(* IEC 61131-3 sources: FB_Sequence/tests, 8 files *)

(* ---- FB_SEQ_ControlMock.st ---- *)
// OFFLINE TEST DOUBLE ONLY. No I/O, equipment logic or safety function.
// Call before FB_Sequence in the same cyclic task: requests take one scan to echo.
FUNCTION_BLOCK FB_SEQ_ControlMock
VAR_INPUT
    xEnable : BOOL := FALSE;
    stRequest : ST_SEQ_CONTROL_REQUEST;
    stConfig : ST_SEQ_CONFIG;
    xAllowRequests : BOOL := FALSE;
    xAllowExecution : BOOL := FALSE;
    xAllowPublication : BOOL := FALSE;
    xQualified : BOOL := FALSE;
    xStepComplete : BOOL := FALSE;
    xFaulted : BOOL := FALSE;
    xRejectRequest : BOOL := FALSE;
    xFinishActions : BOOL := FALSE;
    udiAuthorityID : UDINT := 0;
END_VAR
VAR_OUTPUT
    stAuthority : ST_SEQ_CONTROL_AUTHORITY;
    stResult : ST_SEQ_CONTROL_RESULT;
    stRuntime : ST_SEQ_CONTROL_RUNTIME;
END_VAR
VAR
    stEmptyAuthority : ST_SEQ_CONTROL_AUTHORITY;
    stEmptyResult : ST_SEQ_CONTROL_RESULT;
    stEmptyRuntime : ST_SEQ_CONTROL_RUNTIME;
    xGrantValid : BOOL;
    xRequestMatches : BOOL;
    xOwnerMatches : BOOL;
    xOwned : BOOL;
    xClosureDone : BOOL;
    udiOwnerSession : UDINT;
    uiOwnerProcess : UINT;
    udiOwnerBatch : UDINT;
    udiToken : UDINT;
END_VAR

// Permission loss, disable and authority epoch changes NEVER release ownership.
// Reinitialize this non-retained test instance to reset the entire mock.
stAuthority := stEmptyAuthority;
stResult := stEmptyResult;
stRuntime := stEmptyRuntime;
xGrantValid := xEnable AND (stConfig.udiSessionID > 0)
    AND (stConfig.uiProcessID > 0) AND (udiAuthorityID > 0);
IF xGrantValid THEN
    stAuthority.xValid := TRUE;
    stAuthority.udiSessionID := stConfig.udiSessionID;
    stAuthority.uiProcessID := stConfig.uiProcessID;
    stAuthority.udiAuthorityID := udiAuthorityID;
    stAuthority.udiAgeMs := 0; // Freshly republished on every invocation.
    stAuthority.xAllowRequests := xAllowRequests;
    stAuthority.xAllowExecution := xAllowExecution;
    stAuthority.xAllowPublication := xAllowPublication;

    stRuntime.xValid := TRUE;
    stRuntime.udiSessionID := stConfig.udiSessionID;
    stRuntime.uiProcessID := stConfig.uiProcessID;
    stRuntime.udiAuthorityID := udiAuthorityID;
    stRuntime.udiAgeMs := 0;
    stRuntime.xReady := NOT xFaulted;
    stRuntime.xFaulted := xFaulted;
    stRuntime.udiBatchID := udiOwnerBatch;
END_IF;

xRequestMatches := xGrantValid AND xAllowRequests AND stRequest.xValid
    AND (stRequest.udiSessionID = stConfig.udiSessionID)
    AND (stRequest.uiProcessID = stConfig.uiProcessID)
    AND (stRequest.udiAuthorityID = udiAuthorityID)
    AND (stRequest.udiBatchID > 0) AND (stRequest.udiIntentID > 0);
xOwnerMatches := (stRequest.udiSessionID = udiOwnerSession)
    AND (stRequest.uiProcessID = uiOwnerProcess)
    AND (stRequest.udiBatchID = udiOwnerBatch);

IF xRequestMatches THEN
    stResult.xValid := TRUE;
    stResult.udiSessionID := stRequest.udiSessionID;
    stResult.uiProcessID := stRequest.uiProcessID;
    stResult.udiAuthorityID := stRequest.udiAuthorityID;
    stResult.udiBatchID := stRequest.udiBatchID;
    stResult.udiIntentID := stRequest.udiIntentID;
    stResult.udiAgeMs := 0;
    stRuntime.udiBatchID := stRequest.udiBatchID;
    stRuntime.udiIntentID := stRequest.udiIntentID;
    // Explicit positive handling below; unsupported requests are rejected.
    IF NOT xRejectRequest THEN
        CASE stRequest.eAction OF
        E_SEQ_ACTION.Acquire:
            IF xAllowExecution AND NOT xFaulted AND ((NOT xOwned) OR xOwnerMatches) THEN
                IF NOT xOwned THEN
                    xOwned := TRUE;
                    udiOwnerSession := stRequest.udiSessionID;
                    uiOwnerProcess := stRequest.uiProcessID;
                    udiOwnerBatch := stRequest.udiBatchID;
                    udiToken := 1;
                    xClosureDone := FALSE;
                END_IF;
                stResult.xAccepted := TRUE;
                stResult.xDone := TRUE;
            END_IF;
        E_SEQ_ACTION.Execute:
            IF xAllowExecution AND NOT xFaulted AND xOwned AND xOwnerMatches
               AND (stRequest.udiResourceToken = udiToken) THEN
                stResult.xAccepted := TRUE;
                stRuntime.xQualified := xQualified;
                stRuntime.xStepComplete := xStepComplete;
                // Acceptance never implies step completion or a lifecycle Done.
                xClosureDone := FALSE;
            END_IF;
        E_SEQ_ACTION.Hold:
            IF xOwned AND xOwnerMatches AND (stRequest.udiResourceToken = udiToken) THEN
                stResult.xAccepted := TRUE;
                stResult.xDone := xFinishActions;
                xClosureDone := FALSE; // A confirmed hold is not batch closure.
            END_IF;
        E_SEQ_ACTION.Complete, E_SEQ_ACTION.Stop, E_SEQ_ACTION.Abort:
            IF (NOT xOwned) OR xOwnerMatches THEN
                // Token zero may occur if an Acquire ACK was lost before abort.
                // Session/process/batch still identify the owned transaction.
                stResult.xAccepted := TRUE;
                stResult.xDone := xFinishActions;
                IF xFinishActions THEN
                    xClosureDone := TRUE;
                    udiOwnerSession := stRequest.udiSessionID;
                    uiOwnerProcess := stRequest.uiProcessID;
                    udiOwnerBatch := stRequest.udiBatchID;
                END_IF;
            END_IF;
        E_SEQ_ACTION.Release:
            IF xOwnerMatches AND xClosureDone THEN
                stResult.xAccepted := TRUE;
                stResult.xDone := TRUE;
                xOwned := FALSE;
                udiToken := 0;
                // Preserve closed identity for idempotent repeated Release.
                stResult.xReleased := TRUE;
            END_IF;
        END_CASE;
    END_IF;
    stResult.xRejected := NOT stResult.xAccepted;
    IF stResult.xRejected THEN stResult.uiReasonID := 1; END_IF;
    stResult.xResourceGranted := xOwned;
    stResult.udiResourceToken := udiToken;
END_IF;

IF xGrantValid THEN
    stRuntime.xResourceGranted := xOwned;
    stRuntime.udiResourceToken := udiToken;
END_IF;
END_FUNCTION_BLOCK

(* ---- PRG_SEQ_AuthorityTests.st ---- *)
// OFFLINE CORRELATION REGRESSION, 8 scans. Expected TRUE,8,0,65535 for
// xDone,uiChecks,uiFailures,uiFirstFailureStep. Requires target IDE execution.
// A Release result from authority 1 cannot combine with runtime from authority 2.
PROGRAM PRG_SEQ_AuthorityTests
VAR
    fbSeq : FB_Sequence;
    fbMock : FB_SEQ_ControlMock;
    stConfig : ST_SEQ_CONFIG;
    stRecipe : ST_SEQ_RECIPE;
    stCommand : ST_SEQ_COMMAND_REQUEST;
    stAuthorityToSeq : ST_SEQ_CONTROL_AUTHORITY;
    stRuntimeToSeq : ST_SEQ_CONTROL_RUNTIME;
    udiAuthorityID : UDINT := 1;
    udiReleaseIntentBefore : UDINT;
    xAllowExecution : BOOL := TRUE;
    xFinishActions : BOOL;
    xPass : BOOL;
    uiStep : UINT;
    uiChecks : UINT;
    uiFailures : UINT;
    uiFirstFailureStep : UINT := UINT#65535;
    xDone : BOOL;
END_VAR

IF xDone THEN RETURN; END_IF;
stCommand.xValid := FALSE;
xFinishActions := FALSE;
CASE uiStep OF
0:
    stConfig.uiProcessID := 1;
    stConfig.udiSessionID := 6001;
    stConfig.udiMaxFeedbackAgeMs := 100;
    stConfig.udiTransitionTimeoutMs := 1000;
    stConfig.udiMaxCycleMs := 100;
    stRecipe.udiRecipeID := 10;
    stRecipe.udiRevision := 1;
    stRecipe.uiStepCount := 1;
    stRecipe.astSteps[1].uiStepID := 100;
    stRecipe.astSteps[1].uiPhaseID := 1;
    stRecipe.astSteps[1].uiProfileID := 1;
    stRecipe.astSteps[1].eKind := E_SEQ_STEP_KIND.WaitComplete;
    stRecipe.astSteps[1].udiTimeoutMs := 5000;
    stCommand.udiSessionID := stConfig.udiSessionID;
    stCommand.uiProcessID := 1;
    stCommand.uiSourceID := 1;
    stCommand.udiRecipeID := 10;
    stCommand.udiRecipeRevision := 1;
    stCommand.udiRequestID := 1;
    stCommand.eCommand := E_SEQ_CMD.LoadRecipe;
    stCommand.xValid := TRUE;
1:
    stCommand.udiBatchID := 1;
    stCommand.udiRequestID := 2;
    stCommand.eCommand := E_SEQ_CMD.Start;
    stCommand.xValid := TRUE;
3:
    xAllowExecution := FALSE;
4:
    xFinishActions := TRUE;
5:
    udiReleaseIntentBefore := fbSeq.stControlRequest.udiIntentID;
6:
    udiAuthorityID := 2;
7:
    stCommand.udiRequestID := 3;
    stCommand.eCommand := E_SEQ_CMD.Reset;
    stCommand.xValid := TRUE;
END_CASE;
fbMock(xEnable := TRUE, stRequest := fbSeq.stControlRequest,
    stConfig := stConfig, xAllowRequests := TRUE,
    xAllowExecution := xAllowExecution, xAllowPublication := TRUE,
    xQualified := FALSE, xStepComplete := FALSE,
    xFaulted := FALSE, xRejectRequest := FALSE,
    xFinishActions := xFinishActions, udiAuthorityID := udiAuthorityID);
stAuthorityToSeq := fbMock.stAuthority;
stRuntimeToSeq := fbMock.stRuntime;
IF uiStep = 5 THEN
    // All scalar freshness/BatchID/IntentID fields match, but generations differ.
    // Keep the valid old-generation Release result intact to reproduce the bug.
    stAuthorityToSeq.udiAuthorityID := 2;
    stRuntimeToSeq.udiAuthorityID := 2;
END_IF;
fbSeq(xEnable := TRUE, stConfig := stConfig, udiDeltaMs := 10,
    stCommand := stCommand, stRecipeCandidate := stRecipe,
    stAuthority := stAuthorityToSeq, stControlResult := fbMock.stResult,
    stControlRuntime := stRuntimeToSeq,
    udiEventAckSessionID := 0, udiEventAckID := 0);
xPass := FALSE;
CASE uiStep OF
0:
    xPass := fbSeq.stRuntime.xRecipeLoaded;
1:
    xPass := fbSeq.stRuntime.eState = E_SEQ_STATE.Starting;
2:
    xPass := fbSeq.stRuntime.eState = E_SEQ_STATE.Running;
3:
    xPass := (fbSeq.stRuntime.eState = E_SEQ_STATE.Faulted)
        AND (fbSeq.stControlRequest.eAction = E_SEQ_ACTION.Abort);
4:
    xPass := (fbSeq.stRuntime.eState = E_SEQ_STATE.Faulted)
        AND (fbSeq.stControlRequest.eAction = E_SEQ_ACTION.Release);
5:
    xPass := fbMock.stResult.xReleased AND (fbMock.stResult.udiAuthorityID = 1)
        AND (fbSeq.stRuntime.eState = E_SEQ_STATE.Faulted)
        AND fbSeq.stControlRequest.xValid
        AND (fbSeq.stControlRequest.eAction = E_SEQ_ACTION.Release)
        AND (fbSeq.stControlRequest.udiAuthorityID = 2)
        AND (fbSeq.stControlRequest.udiIntentID > udiReleaseIntentBefore);
6:
    xPass := fbMock.stResult.xReleased AND (fbMock.stResult.udiAuthorityID = 2)
        AND (fbSeq.stRuntime.eState = E_SEQ_STATE.Faulted)
        AND NOT fbSeq.stControlRequest.xValid;
7:
    xPass := (fbSeq.stRuntime.eState = E_SEQ_STATE.Idle)
        AND (fbSeq.stCommandResult.eResult = E_SEQ_RESULT.Accepted);
END_CASE;
uiChecks := uiChecks + 1;
IF NOT xPass THEN
    uiFailures := uiFailures + 1;
    IF uiFirstFailureStep = UINT#65535 THEN uiFirstFailureStep := uiStep; END_IF;
END_IF;
IF uiStep >= 7 THEN xDone := TRUE;
ELSE uiStep := uiStep + 1; END_IF;
END_PROGRAM

(* ---- PRG_SEQ_Demo.st ---- *)
PROGRAM PRG_SEQ_Demo
VAR
    // Offline-only sandbox. Both mock and Sequence begin disabled.
    xControlMockEnabled : BOOL := FALSE;
    xSequenceEnabled : BOOL := FALSE;
    xAllowRequests : BOOL := FALSE;
    xAllowExecution : BOOL := FALSE;
    xAllowPublication : BOOL := FALSE;
    xQualified : BOOL := FALSE;
    xStepComplete : BOOL := FALSE;
    xFaulted : BOOL := FALSE;
    xRejectRequest : BOOL := FALSE;
    xFinishActions : BOOL := FALSE;
    udiAuthorityID : UDINT := 1;
    stConfig : ST_SEQ_CONFIG := (uiProcessID := 1, udiSessionID := 1,
        udiMaxFeedbackAgeMs := 250, udiTransitionTimeoutMs := 5000, udiMaxCycleMs := 100);
    stCommand : ST_SEQ_COMMAND_REQUEST;
    stRecipe : ST_SEQ_RECIPE;
    udiAckSessionID : UDINT;
    udiAckEventID : UDINT;
    fbControlMock : FB_SEQ_ControlMock;
    fbSequence : FB_Sequence;
    xInitialized : BOOL;
END_VAR

IF NOT xInitialized THEN
    xInitialized := TRUE;
    stRecipe.udiRecipeID := 1;
    stRecipe.udiRevision := 1;
    stRecipe.uiStepCount := 3;
    stRecipe.astSteps[1].uiStepID := 10;
    stRecipe.astSteps[1].uiPhaseID := 10;
    stRecipe.astSteps[1].uiProfileID := 100;
    stRecipe.astSteps[1].eKind := E_SEQ_STEP_KIND.WaitQualified;
    stRecipe.astSteps[1].udiQualifiedMs := 250;
    stRecipe.astSteps[1].udiTimeoutMs := 10000;
    stRecipe.astSteps[2].uiStepID := 20;
    stRecipe.astSteps[2].uiPhaseID := 20;
    stRecipe.astSteps[2].uiProfileID := 200;
    stRecipe.astSteps[2].eKind := E_SEQ_STEP_KIND.WaitComplete;
    stRecipe.astSteps[2].udiTimeoutMs := 10000;
    stRecipe.astSteps[3].uiStepID := 30;
    stRecipe.astSteps[3].uiPhaseID := 30;
    stRecipe.astSteps[3].uiProfileID := 300;
    stRecipe.astSteps[3].eKind := E_SEQ_STEP_KIND.WaitOperator;
    stRecipe.astSteps[3].udiTimeoutMs := 10000;
END_IF;

// One task, one call per scan, previous request consumed by mock on next scan.
fbControlMock(xEnable := xControlMockEnabled, stRequest := fbSequence.stControlRequest,
    stConfig := stConfig, xAllowRequests := xAllowRequests, xAllowExecution := xAllowExecution,
    xAllowPublication := xAllowPublication, xQualified := xQualified,
    xStepComplete := xStepComplete, xFaulted := xFaulted, xRejectRequest := xRejectRequest,
    xFinishActions := xFinishActions, udiAuthorityID := udiAuthorityID);
fbSequence(xEnable := xSequenceEnabled, stConfig := stConfig, udiDeltaMs := 20,
    stCommand := stCommand, stRecipeCandidate := stRecipe,
    stAuthority := fbControlMock.stAuthority, stControlResult := fbControlMock.stResult,
    stControlRuntime := fbControlMock.stRuntime,
    udiEventAckSessionID := udiAckSessionID, udiEventAckID := udiAckEventID);
// 20 ms here is synthetic simulation time, not a claim of measured target timing.
END_PROGRAM

(* ---- PRG_SEQ_IntegrationTests.st ---- *)
// OFFLINE MULTISCAN TEST POU: import with production types/FBs and ControlMock.
// Assign ONLY to a simulator/test task with no physical I/O. Every call is 10 ms
// of simulated time. Fresh non-retained instances run 28 checks in 28 calls.
// Inspect xDone, uiChecks, uiFailures, uiFirstFailureStep. Expected: TRUE,28,0,65535.
// Reinitialize the application to rerun; changing uiStep alone is insufficient.
// These are executable IDE test scenarios; their presence is not a test-run claim.
PROGRAM PRG_SEQ_IntegrationTests
VAR
    fbSeq : FB_Sequence;
    fbMock : FB_SEQ_ControlMock;
    stConfig : ST_SEQ_CONFIG;
    stRecipe : ST_SEQ_RECIPE;
    stCommand : ST_SEQ_COMMAND_REQUEST;
    stResultToSeq : ST_SEQ_CONTROL_RESULT;
    stRuntimeToSeq : ST_SEQ_CONTROL_RUNTIME;
    xMockEnable : BOOL;
    xAllowRequests : BOOL;
    xAllowExecution : BOOL;
    xAllowPublication : BOOL;
    xQualified : BOOL;
    xStepComplete : BOOL;
    xFinishActions : BOOL;
    udiAuthorityID : UDINT;
    xCorruptResultID : BOOL;
    xCorruptRuntimeID : BOOL;
    xPass : BOOL;
    uiStep : UINT;
    uiChecks : UINT;
    uiFailures : UINT;
    uiFirstFailureStep : UINT := UINT#65535;
    xDone : BOOL;
END_VAR

IF xDone THEN RETURN; END_IF;

// Default stimuli are inert; permission changes remain in effect across scans.
stCommand.xValid := FALSE;
xQualified := FALSE;
xStepComplete := FALSE;
xFinishActions := FALSE;
xCorruptResultID := FALSE;
xCorruptRuntimeID := FALSE;

CASE uiStep OF
0: // Neither mock enable nor a Control grant exists.
    stConfig.uiProcessID := 1;
    stConfig.udiSessionID := 1001;
    stConfig.udiMaxFeedbackAgeMs := 100;
    stConfig.udiTransitionTimeoutMs := 1000;
    stConfig.udiMaxCycleMs := 100;
    stRecipe.udiRecipeID := 10;
    stRecipe.udiRevision := 1;
    stRecipe.uiStepCount := 1;
    stRecipe.astSteps[1].uiStepID := 100;
    stRecipe.astSteps[1].uiPhaseID := 1;
    stRecipe.astSteps[1].uiProfileID := 1;
    stRecipe.astSteps[1].eKind := E_SEQ_STEP_KIND.WaitQualified;
    stRecipe.astSteps[1].udiQualifiedMs := 30;
    stRecipe.astSteps[1].udiTimeoutMs := 2000;
    stCommand.udiSessionID := stConfig.udiSessionID;
    stCommand.uiProcessID := stConfig.uiProcessID;
    stCommand.uiSourceID := 1;
    stCommand.udiRecipeID := stRecipe.udiRecipeID;
    stCommand.udiRecipeRevision := stRecipe.udiRevision;
    stCommand.udiRequestID := 1;
    stCommand.eCommand := E_SEQ_CMD.LoadRecipe;
    stCommand.xValid := TRUE;
1: // Permission bits alone cannot manufacture a nonzero Control authority.
    xMockEnable := TRUE;
    xAllowRequests := TRUE;
    xAllowExecution := TRUE;
    xAllowPublication := TRUE;
2: // A new request ID is required after the denied request.
    udiAuthorityID := 1;
    stCommand.udiRequestID := 2;
    stCommand.eCommand := E_SEQ_CMD.LoadRecipe;
    stCommand.xValid := TRUE;
3:
    stCommand.udiRequestID := 3;
    stCommand.eCommand := E_SEQ_CMD.Start;
    stCommand.udiBatchID := 1;
    stCommand.xValid := TRUE;
4: // Acquire has completed in Control, but an unrelated ACK cannot advance.
    xCorruptResultID := TRUE;
5: // The original matching Acquire result is now admitted.
    ;
6: // A matching accepted result plus unrelated runtime is still insufficient.
    xQualified := TRUE;
    xStepComplete := TRUE;
    xCorruptRuntimeID := TRUE;
7: // First qualified observation establishes the interval boundary.
    xQualified := TRUE;
8: // An unqualified interval must not accrue qualified time.
    xQualified := FALSE;
9, 10, 11, 12:
    xQualified := TRUE;
13: // Control accepted Complete, but has not finished the physical closure.
    ;
14:
    xFinishActions := TRUE;
15: // Release is a separate transaction after closure Done.
    ;
16:
    stCommand.udiRequestID := 4;
    stCommand.eCommand := E_SEQ_CMD.Reset;
    stCommand.xValid := TRUE;
17:
    stCommand.udiRequestID := 5;
    stCommand.eCommand := E_SEQ_CMD.Start;
    stCommand.udiBatchID := 2;
    stCommand.xValid := TRUE;
18:
    ;
19: // Revoke requests and execution during the second batch.
    xAllowRequests := FALSE;
    xAllowExecution := FALSE;
20: // Restoring both permissions cannot resume the faulted batch.
    xAllowRequests := TRUE;
    xAllowExecution := TRUE;
21: // Publication permission controls every public Service envelope.
    xAllowPublication := FALSE;
22: // Requests remain permitted for closure while execution is denied.
    xAllowPublication := TRUE;
    xAllowExecution := FALSE;
23: // New Control epoch must not silently erase existing ownership.
    udiAuthorityID := 2;
24:
    xFinishActions := TRUE;
25:
    ;
26: // Reset requires the confirmed Abort then Release, not just a new grant.
    stCommand.udiRequestID := 6;
    stCommand.eCommand := E_SEQ_CMD.Reset;
    stCommand.xValid := TRUE;
27: // Request permission does not imply permission to start execution.
    stCommand.udiRequestID := 7;
    stCommand.eCommand := E_SEQ_CMD.Start;
    stCommand.udiBatchID := 3;
    stCommand.xValid := TRUE;
END_CASE;

// One scan of request/feedback latency, with fresh snapshots on every mock call.
fbMock(xEnable := xMockEnable, stRequest := fbSeq.stControlRequest,
    stConfig := stConfig, xAllowRequests := xAllowRequests,
    xAllowExecution := xAllowExecution, xAllowPublication := xAllowPublication,
    xQualified := xQualified, xStepComplete := xStepComplete,
    xFaulted := FALSE, xRejectRequest := FALSE,
    xFinishActions := xFinishActions, udiAuthorityID := udiAuthorityID);
stResultToSeq := fbMock.stResult;
stRuntimeToSeq := fbMock.stRuntime;
IF xCorruptResultID THEN
    stResultToSeq.udiIntentID := stResultToSeq.udiIntentID + 100;
END_IF;
IF xCorruptRuntimeID THEN
    stRuntimeToSeq.udiIntentID := stRuntimeToSeq.udiIntentID + 100;
END_IF;
fbSeq(xEnable := TRUE, stConfig := stConfig, udiDeltaMs := 10,
    stCommand := stCommand, stRecipeCandidate := stRecipe,
    stAuthority := fbMock.stAuthority, stControlResult := stResultToSeq,
    stControlRuntime := stRuntimeToSeq,
    udiEventAckSessionID := 0, udiEventAckID := 0);

xPass := FALSE;
CASE uiStep OF
0, 1:
    xPass := NOT fbSeq.stControlRequest.xValid
        AND NOT fbSeq.stRuntime.xDataValid AND NOT fbSeq.stCommandResult.xValid
        AND NOT fbSeq.xEventAvailable AND (fbSeq.uiEventCount = 0)
        AND (fbSeq.stRuntime.udiSessionID = 0) AND (fbSeq.stEvent.udiEventID = 0);
2:
    xPass := fbSeq.stRuntime.xDataValid AND fbSeq.stRuntime.xRecipeLoaded
        AND (fbSeq.stRuntime.eState = E_SEQ_STATE.Idle)
        AND (fbSeq.stCommandResult.eResult = E_SEQ_RESULT.Accepted)
        AND (fbSeq.stCommandResult.udiRequestID = 2);
3:
    xPass := (fbSeq.stRuntime.eState = E_SEQ_STATE.Starting)
        AND (fbSeq.stControlRequest.eAction = E_SEQ_ACTION.Acquire)
        AND fbSeq.stControlRequest.xValid;
4:
    xPass := fbMock.stResult.xDone AND fbMock.stRuntime.xResourceGranted
        AND (fbSeq.stRuntime.eState = E_SEQ_STATE.Starting)
        AND (fbSeq.stRuntime.udiResourceToken = 0)
        AND (fbSeq.stControlRequest.eAction = E_SEQ_ACTION.Acquire);
5:
    xPass := (fbSeq.stRuntime.eState = E_SEQ_STATE.Running)
        AND (fbSeq.stControlRequest.eAction = E_SEQ_ACTION.Execute)
        AND (fbSeq.stRuntime.udiResourceToken = 1);
6:
    xPass := fbMock.stResult.xAccepted AND NOT fbMock.stResult.xDone
        AND (fbSeq.stRuntime.eState = E_SEQ_STATE.Running)
        AND (fbSeq.stRuntime.udiQualifiedElapsedMs = 0);
7, 8, 9:
    xPass := (fbSeq.stRuntime.eState = E_SEQ_STATE.Running)
        AND (fbSeq.stRuntime.udiQualifiedElapsedMs = 0);
10:
    xPass := (fbSeq.stRuntime.eState = E_SEQ_STATE.Running)
        AND (fbSeq.stRuntime.udiQualifiedElapsedMs = 10);
11:
    xPass := (fbSeq.stRuntime.eState = E_SEQ_STATE.Running)
        AND (fbSeq.stRuntime.udiQualifiedElapsedMs = 20);
12:
    xPass := (fbSeq.stRuntime.eState = E_SEQ_STATE.Completing)
        AND (fbSeq.stControlRequest.eAction = E_SEQ_ACTION.Complete)
        AND (fbSeq.stRuntime.udiQualifiedElapsedMs = 30)
        AND fbMock.stRuntime.xResourceGranted;
13:
    xPass := fbMock.stResult.xAccepted AND NOT fbMock.stResult.xDone
        AND (fbSeq.stRuntime.eState = E_SEQ_STATE.Completing)
        AND (fbSeq.stControlRequest.eAction = E_SEQ_ACTION.Complete)
        AND fbMock.stRuntime.xResourceGranted;
14:
    xPass := fbMock.stResult.xDone
        AND (fbSeq.stRuntime.eState = E_SEQ_STATE.Completing)
        AND (fbSeq.stControlRequest.eAction = E_SEQ_ACTION.Release)
        AND fbMock.stRuntime.xResourceGranted;
15:
    xPass := fbMock.stResult.xReleased AND NOT fbMock.stRuntime.xResourceGranted
        AND (fbSeq.stRuntime.eState = E_SEQ_STATE.Complete)
        AND (fbSeq.stRuntime.udiResourceToken = 0)
        AND NOT fbSeq.stControlRequest.xValid;
16:
    xPass := (fbSeq.stRuntime.eState = E_SEQ_STATE.Idle)
        AND (fbSeq.stRuntime.udiBatchID = 0)
        AND (fbSeq.stCommandResult.eResult = E_SEQ_RESULT.Accepted);
17:
    xPass := (fbSeq.stRuntime.eState = E_SEQ_STATE.Starting)
        AND (fbSeq.stRuntime.udiBatchID = 2)
        AND (fbSeq.stControlRequest.eAction = E_SEQ_ACTION.Acquire);
18:
    xPass := (fbSeq.stRuntime.eState = E_SEQ_STATE.Running)
        AND (fbSeq.stControlRequest.eAction = E_SEQ_ACTION.Execute)
        AND fbMock.stRuntime.xResourceGranted;
19:
    xPass := (fbSeq.stRuntime.eState = E_SEQ_STATE.Faulted)
        AND (fbSeq.stRuntime.eReason = E_SEQ_REASON.AuthorityDenied)
        AND NOT fbSeq.stControlRequest.xValid AND NOT fbMock.stResult.xValid
        AND fbMock.stRuntime.xResourceGranted;
20:
    xPass := (fbSeq.stRuntime.eState = E_SEQ_STATE.Faulted)
        AND fbSeq.stControlRequest.xValid
        AND (fbSeq.stControlRequest.eAction = E_SEQ_ACTION.Abort)
        AND fbMock.stRuntime.xResourceGranted;
21:
    xPass := NOT fbSeq.stRuntime.xDataValid AND NOT fbSeq.stCommandResult.xValid
        AND (fbSeq.stRuntime.udiSessionID = 0) AND (fbSeq.stRuntime.udiBatchID = 0)
        AND (fbSeq.stCommandResult.udiRequestID = 0)
        AND NOT fbSeq.xEventAvailable AND (fbSeq.stEvent.udiEventID = 0)
        AND (fbSeq.uiEventCount = 0) AND (fbSeq.udiEventsDropped = 0)
        AND (fbSeq.stControlRequest.eAction = E_SEQ_ACTION.Abort)
        AND fbMock.stRuntime.xResourceGranted;
22:
    xPass := (fbSeq.stRuntime.eState = E_SEQ_STATE.Faulted)
        AND (fbSeq.stControlRequest.eAction = E_SEQ_ACTION.Abort)
        AND fbSeq.xEventAvailable AND fbMock.stRuntime.xResourceGranted;
23:
    xPass := (fbSeq.stRuntime.eState = E_SEQ_STATE.Faulted)
        AND (fbSeq.stControlRequest.eAction = E_SEQ_ACTION.Abort)
        AND (fbSeq.stControlRequest.udiAuthorityID = 2)
        AND NOT fbMock.stResult.xValid AND fbMock.stRuntime.xResourceGranted;
24:
    xPass := (fbSeq.stRuntime.eState = E_SEQ_STATE.Faulted)
        AND fbMock.stResult.xDone AND (fbSeq.stControlRequest.eAction = E_SEQ_ACTION.Release)
        AND fbMock.stRuntime.xResourceGranted;
25:
    xPass := (fbSeq.stRuntime.eState = E_SEQ_STATE.Faulted)
        AND fbMock.stResult.xReleased AND NOT fbMock.stRuntime.xResourceGranted
        AND NOT fbSeq.stControlRequest.xValid AND (fbSeq.stRuntime.udiResourceToken = 0);
26:
    xPass := (fbSeq.stRuntime.eState = E_SEQ_STATE.Idle)
        AND (fbSeq.stCommandResult.eResult = E_SEQ_RESULT.Accepted)
        AND NOT fbMock.stRuntime.xResourceGranted;
27:
    xPass := (fbSeq.stRuntime.eState = E_SEQ_STATE.Idle)
        AND (fbSeq.stCommandResult.eResult = E_SEQ_RESULT.Rejected)
        AND (fbSeq.stCommandResult.eReason = E_SEQ_REASON.AuthorityDenied)
        AND NOT fbSeq.stControlRequest.xValid;
END_CASE;

uiChecks := uiChecks + 1;
IF NOT xPass THEN
    IF uiFailures = 0 THEN uiFirstFailureStep := uiStep; END_IF;
    uiFailures := uiFailures + 1;
END_IF;
IF uiStep = 27 THEN xDone := TRUE;
ELSE uiStep := uiStep + 1; END_IF;
END_PROGRAM

(* ---- PRG_SEQ_LifecycleTests.st ---- *)
// OFFLINE MULTISCAN TEST ONLY: no physical I/O or task scheduling assumptions.
// Run a fresh, non-retained instance for 56 simulated scans of 10 ms each.
// Expected: xDone=TRUE, uiChecks=56, uiFailures=0, uiFirstFailureStep=65535.
// Exercises actual FB_Sequence code when run in the target IDE; NOT run here.
PROGRAM PRG_SEQ_LifecycleTests
VAR
    fbSeq : FB_Sequence;
    fbMock : FB_SEQ_ControlMock;
    stConfig : ST_SEQ_CONFIG;
    stRecipe : ST_SEQ_RECIPE;
    stCommand : ST_SEQ_COMMAND_REQUEST;
    stRuntimeToSeq : ST_SEQ_CONTROL_RUNTIME;
    xQualified : BOOL;
    xFinishActions : BOOL;
    xInjectHoldQualified : BOOL;
    xInjectNotReady : BOOL;
    xPass : BOOL;
    xSawResetBatch : BOOL;
    udiRequestID : UDINT;
    udiAck : UDINT;
    udiPrompt : UDINT;
    uiStep : UINT;
    uiChecks : UINT;
    uiFailures : UINT;
    uiFirstFailureStep : UINT := UINT#65535;
    xDone : BOOL;
END_VAR

IF xDone THEN RETURN; END_IF;
stCommand.xValid := FALSE;
xQualified := TRUE;
xFinishActions := FALSE;
xInjectHoldQualified := FALSE;
xInjectNotReady := FALSE;

CASE uiStep OF
0:
    stConfig.uiProcessID := 1;
    stConfig.udiSessionID := 5001;
    stConfig.udiMaxFeedbackAgeMs := 100;
    stConfig.udiTransitionTimeoutMs := 30;
    stConfig.udiMaxCycleMs := 100;
    stRecipe.udiRecipeID := 10;
    stRecipe.udiRevision := 1;
    stRecipe.uiStepCount := 1;
    stRecipe.astSteps[1].uiStepID := 100;
    stRecipe.astSteps[1].uiPhaseID := 1;
    stRecipe.astSteps[1].uiProfileID := 1;
    stRecipe.astSteps[1].eKind := E_SEQ_STEP_KIND.WaitQualified;
    stRecipe.astSteps[1].udiQualifiedMs := 100;
    stRecipe.astSteps[1].udiTimeoutMs := 5000;
    stCommand.udiSessionID := stConfig.udiSessionID;
    stCommand.uiProcessID := stConfig.uiProcessID;
    stCommand.uiSourceID := 1;
    stCommand.udiRecipeID := 10;
    stCommand.udiRecipeRevision := 1;
    stCommand.eCommand := E_SEQ_CMD.LoadRecipe;
    stCommand.xValid := TRUE;
1:
    stCommand.udiBatchID := 1;
    stCommand.eCommand := E_SEQ_CMD.Start;
    stCommand.xValid := TRUE;
5:
    stCommand.eCommand := E_SEQ_CMD.Hold;
    stCommand.xValid := TRUE;
6:
    xFinishActions := TRUE;
7:
    xInjectHoldQualified := TRUE;
8: // Old Hold feedback must not qualify the first interval after Resume.
    xInjectHoldQualified := TRUE;
    stCommand.eCommand := E_SEQ_CMD.Resume;
    stCommand.xValid := TRUE;
9: // Changing the candidate cannot mutate the already applied recipe snapshot.
    stRecipe.udiRevision := 99;
    stRecipe.astSteps[1].udiQualifiedMs := 1;
11:
    stCommand.eCommand := E_SEQ_CMD.Stop;
    stCommand.xValid := TRUE;
13:
    xFinishActions := TRUE;
15:
    stCommand.eCommand := E_SEQ_CMD.Reset;
    stCommand.xValid := TRUE;
16:
    stRecipe.udiRevision := 2;
    stRecipe.astSteps[1].eKind := E_SEQ_STEP_KIND.WaitOperator;
    stRecipe.astSteps[1].udiQualifiedMs := 0;
    stCommand.udiRecipeRevision := 2;
    stCommand.eCommand := E_SEQ_CMD.LoadRecipe;
    stCommand.xValid := TRUE;
17:
    stCommand.udiBatchID := 2;
    stCommand.eCommand := E_SEQ_CMD.Start;
    stCommand.xValid := TRUE;
19: // Matching/qualified feedback that is not Ready must reject confirmation.
    udiPrompt := fbSeq.stRuntime.udiPromptID;
    stCommand.uiStepID := 100;
    stCommand.udiPromptID := udiPrompt;
    stCommand.eCommand := E_SEQ_CMD.ConfirmStep;
    stCommand.xValid := TRUE;
    xInjectNotReady := TRUE;
20:
    stCommand.udiPromptID := udiPrompt + 1;
    stCommand.eCommand := E_SEQ_CMD.ConfirmStep;
    stCommand.xValid := TRUE;
26: // Running now exceeds the transition limit; new Completing starts at zero.
    stCommand.udiPromptID := udiPrompt;
    stCommand.eCommand := E_SEQ_CMD.ConfirmStep;
    stCommand.xValid := TRUE;
27:
    xFinishActions := TRUE;
29:
    stCommand.eCommand := E_SEQ_CMD.Reset;
    stCommand.xValid := TRUE;
30:
    stCommand.udiBatchID := 3;
    stCommand.eCommand := E_SEQ_CMD.Start;
    stCommand.xValid := TRUE;
32:
    stCommand.eCommand := E_SEQ_CMD.Abort;
    stCommand.xValid := TRUE;
33:
    xFinishActions := TRUE;
35:
    stCommand.eCommand := E_SEQ_CMD.Reset;
    stCommand.xValid := TRUE;
36:
    stCommand.udiBatchID := 4;
    stCommand.eCommand := E_SEQ_CMD.Start;
    stCommand.xValid := TRUE;
38:
    stCommand.eCommand := E_SEQ_CMD.Hold;
    stCommand.xValid := TRUE;
42:
    xFinishActions := TRUE;
44:
    stCommand.eCommand := E_SEQ_CMD.Reset;
    stCommand.xValid := TRUE;
END_CASE;
IF stCommand.xValid THEN
    udiRequestID := udiRequestID + 1;
    stCommand.udiRequestID := udiRequestID;
END_IF;

// Acknowledge ONLY an event actually observed in the previous published scan.
udiAck := 0;
IF fbSeq.xEventAvailable THEN
    udiAck := fbSeq.stEvent.udiEventID;
    IF (fbSeq.stEvent.eKind = E_SEQ_EVENT_KIND.CommandResult)
       AND (fbSeq.stEvent.eCommand = E_SEQ_CMD.Reset)
       AND (fbSeq.stEvent.udiBatchID = 1)
       AND (fbSeq.stEvent.eCommandResult = E_SEQ_RESULT.Accepted) THEN
        xSawResetBatch := TRUE;
    END_IF;
END_IF;
fbMock(xEnable := TRUE, stRequest := fbSeq.stControlRequest,
    stConfig := stConfig, xAllowRequests := TRUE,
    xAllowExecution := TRUE, xAllowPublication := TRUE,
    xQualified := xQualified, xStepComplete := FALSE,
    xFaulted := FALSE, xRejectRequest := FALSE,
    xFinishActions := xFinishActions, udiAuthorityID := 1);
stRuntimeToSeq := fbMock.stRuntime;
IF xInjectHoldQualified THEN stRuntimeToSeq.xQualified := TRUE; END_IF;
IF xInjectNotReady THEN stRuntimeToSeq.xReady := FALSE; END_IF;
fbSeq(xEnable := TRUE, stConfig := stConfig, udiDeltaMs := 10,
    stCommand := stCommand, stRecipeCandidate := stRecipe,
    stAuthority := fbMock.stAuthority, stControlResult := fbMock.stResult,
    stControlRuntime := stRuntimeToSeq,
    udiEventAckSessionID := stConfig.udiSessionID, udiEventAckID := udiAck);

xPass := FALSE;
CASE uiStep OF
0:
    xPass := fbSeq.stRuntime.xRecipeLoaded
        AND (fbSeq.stCommandResult.eResult = E_SEQ_RESULT.Accepted);
1, 17, 30, 36:
    xPass := (fbSeq.stRuntime.eState = E_SEQ_STATE.Starting)
        AND (fbSeq.stControlRequest.eAction = E_SEQ_ACTION.Acquire);
2, 3:
    xPass := (fbSeq.stRuntime.eState = E_SEQ_STATE.Running)
        AND (fbSeq.stRuntime.udiQualifiedElapsedMs = 0);
4:
    xPass := (fbSeq.stRuntime.eState = E_SEQ_STATE.Running)
        AND (fbSeq.stRuntime.udiQualifiedElapsedMs = 10);
5:
    xPass := (fbSeq.stRuntime.eState = E_SEQ_STATE.Holding)
        AND (fbSeq.stRuntime.udiQualifiedElapsedMs = 10);
6, 7:
    xPass := (fbSeq.stRuntime.eState = E_SEQ_STATE.Held)
        AND (fbSeq.stRuntime.udiQualifiedElapsedMs = 10);
8, 9:
    xPass := (fbSeq.stRuntime.eState = E_SEQ_STATE.Running)
        AND (fbSeq.stRuntime.udiQualifiedElapsedMs = 10)
        AND (fbSeq.stRuntime.udiRecipeRevision = 1);
10:
    xPass := (fbSeq.stRuntime.eState = E_SEQ_STATE.Running)
        AND (fbSeq.stRuntime.udiQualifiedElapsedMs = 20);
11, 12:
    xPass := (fbSeq.stRuntime.eState = E_SEQ_STATE.Stopping)
        AND (fbSeq.stControlRequest.eAction = E_SEQ_ACTION.Stop);
13:
    xPass := (fbSeq.stRuntime.eState = E_SEQ_STATE.Stopping)
        AND (fbSeq.stControlRequest.eAction = E_SEQ_ACTION.Release);
14:
    xPass := (fbSeq.stRuntime.eState = E_SEQ_STATE.Stopped)
        AND NOT fbSeq.stControlRequest.xValid;
15, 29, 35, 44:
    xPass := (fbSeq.stRuntime.eState = E_SEQ_STATE.Idle)
        AND (fbSeq.stRuntime.udiBatchID = 0)
        AND (fbSeq.stCommandResult.eResult = E_SEQ_RESULT.Accepted);
16:
    xPass := fbSeq.stRuntime.xRecipeLoaded AND (fbSeq.stRuntime.udiRecipeRevision = 2);
18, 21, 22, 23, 24, 25, 31, 37:
    xPass := (fbSeq.stRuntime.eState = E_SEQ_STATE.Running)
        AND fbSeq.stRuntime.xWaitingOperator AND (fbSeq.stRuntime.udiPromptID > 0);
19, 20:
    xPass := (fbSeq.stRuntime.eState = E_SEQ_STATE.Running)
        AND (fbSeq.stCommandResult.eResult = E_SEQ_RESULT.Rejected)
        AND (fbSeq.stCommandResult.eReason = E_SEQ_REASON.InvalidConfirm);
26:
    xPass := (fbSeq.stRuntime.eState = E_SEQ_STATE.Completing)
        AND (fbSeq.stControlRequest.eAction = E_SEQ_ACTION.Complete)
        AND (fbSeq.stRuntime.udiStateElapsedMs = 0)
        AND (fbSeq.stRuntime.eReason = E_SEQ_REASON.None);
27:
    xPass := (fbSeq.stRuntime.eState = E_SEQ_STATE.Completing)
        AND (fbSeq.stControlRequest.eAction = E_SEQ_ACTION.Release);
28:
    xPass := (fbSeq.stRuntime.eState = E_SEQ_STATE.Complete)
        AND NOT fbSeq.stControlRequest.xValid;
32:
    xPass := (fbSeq.stRuntime.eState = E_SEQ_STATE.Aborting)
        AND (fbSeq.stControlRequest.eAction = E_SEQ_ACTION.Abort);
33:
    xPass := (fbSeq.stRuntime.eState = E_SEQ_STATE.Aborting)
        AND (fbSeq.stControlRequest.eAction = E_SEQ_ACTION.Release);
34:
    xPass := (fbSeq.stRuntime.eState = E_SEQ_STATE.Aborted)
        AND NOT fbSeq.stControlRequest.xValid;
38, 39, 40:
    xPass := (fbSeq.stRuntime.eState = E_SEQ_STATE.Holding)
        AND (fbSeq.stControlRequest.eAction = E_SEQ_ACTION.Hold);
41:
    xPass := (fbSeq.stRuntime.eState = E_SEQ_STATE.Faulted)
        AND (fbSeq.stRuntime.eReason = E_SEQ_REASON.TransitionTimeout)
        AND (fbSeq.stControlRequest.eAction = E_SEQ_ACTION.Abort);
42:
    xPass := (fbSeq.stRuntime.eState = E_SEQ_STATE.Faulted)
        AND (fbSeq.stControlRequest.eAction = E_SEQ_ACTION.Release);
43:
    xPass := (fbSeq.stRuntime.eState = E_SEQ_STATE.Faulted)
        AND NOT fbSeq.stControlRequest.xValid
        AND NOT fbMock.stRuntime.xResourceGranted;
ELSE
    xPass := (fbSeq.stRuntime.eState = E_SEQ_STATE.Idle)
        AND (fbSeq.udiEventsDropped = 0);
END_CASE;
IF uiStep = 55 THEN
    xPass := xPass AND xSawResetBatch AND NOT fbSeq.xEventAvailable;
END_IF;
uiChecks := uiChecks + 1;
IF NOT xPass THEN
    uiFailures := uiFailures + 1;
    IF uiFirstFailureStep = UINT#65535 THEN uiFirstFailureStep := uiStep; END_IF;
END_IF;
IF uiStep >= 55 THEN xDone := TRUE;
ELSE uiStep := uiStep + 1; END_IF;
END_PROGRAM

(* ---- PRG_SEQ_SupportTests.st ---- *)
// Simulator-only self-checking POU; no GVLs, physical I/O, network, or tasks.
// Import DUTs, F_SEQ_AddMs, FB_SEQ_* and this PROGRAM into Machine Expert.
// Attach ONLY this POU to a simulator task; observe xDone, uiChecks, uiFailures.
// Expected result: xDone = TRUE, uiChecks = 40, uiFailures = 0.
// Reset/reinitialize the application to rerun: stateful instances are intentional.
// Deliberate sequential FB calls model scan boundaries with explicit deltas.
// These are authored executable simulator tests; not proof of a native compile.
PROGRAM PRG_SEQ_SupportTests
VAR
    xDone : BOOL;
    uiChecks : UINT;
    uiFailures : UINT;
    fbTimer : FB_SEQ_QualifiedTimer;
    fbRecipe : FB_SEQ_RecipeValidator;
    fbQueue : FB_SEQ_EventQueue;
    fbGate : FB_SEQ_CommandGate;
    stRecipe : ST_SEQ_RECIPE;
    stEvent : ST_SEQ_EVENT;
    stCommand : ST_SEQ_COMMAND_REQUEST;
    uiIndex : UINT;
    udiExpectedID : UDINT;
    xDrainCorrect : BOOL;
END_VAR

IF xDone THEN RETURN; END_IF;

// 01 - Overflow-safe addition, including boundary equality.
uiChecks := uiChecks + 1;
IF F_SEQ_AddMs(UDINT#4294967294, UDINT#1) <> UDINT#4294967295 THEN
    uiFailures := uiFailures + 1;
END_IF;
uiChecks := uiChecks + 1;
IF F_SEQ_AddMs(UDINT#4294967294, UDINT#2) <> UDINT#4294967295 THEN
    uiFailures := uiFailures + 1;
END_IF;
uiChecks := uiChecks + 1;
IF F_SEQ_AddMs(UDINT#4294967295, UDINT#4294967295) <> UDINT#4294967295 THEN
    uiFailures := uiFailures + 1;
END_IF;

// 02 - Qualified timer: reset dominates an enabled/qualified call.
fbTimer(xReset := TRUE, xEnable := TRUE, xQualified := TRUE,
    udiDeltaMs := 100, udiTargetMs := 100);
uiChecks := uiChecks + 1;
IF (fbTimer.udiElapsedMs <> 0) OR fbTimer.xDone THEN
    uiFailures := uiFailures + 1;
END_IF;
fbTimer(xReset := FALSE, xEnable := TRUE, xQualified := TRUE,
    udiDeltaMs := 40, udiTargetMs := 100);
uiChecks := uiChecks + 1;
IF (fbTimer.udiElapsedMs <> 40) OR fbTimer.xDone THEN
    uiFailures := uiFailures + 1;
END_IF;
fbTimer(xReset := FALSE, xEnable := FALSE, xQualified := TRUE,
    udiDeltaMs := 80, udiTargetMs := 100);
uiChecks := uiChecks + 1;
IF (fbTimer.udiElapsedMs <> 40) OR fbTimer.xDone THEN
    uiFailures := uiFailures + 1;
END_IF;
fbTimer(xReset := FALSE, xEnable := TRUE, xQualified := FALSE,
    udiDeltaMs := 80, udiTargetMs := 100);
uiChecks := uiChecks + 1;
IF (fbTimer.udiElapsedMs <> 40) OR fbTimer.xDone THEN
    uiFailures := uiFailures + 1;
END_IF;
fbTimer(xReset := FALSE, xEnable := TRUE, xQualified := TRUE,
    udiDeltaMs := UDINT#4294967295, udiTargetMs := 100);
uiChecks := uiChecks + 1;
IF (fbTimer.udiElapsedMs <> 100) OR NOT fbTimer.xDone THEN
    uiFailures := uiFailures + 1;
END_IF;
fbTimer(xReset := FALSE, xEnable := FALSE, xQualified := FALSE,
    udiDeltaMs := 100, udiTargetMs := 100);
uiChecks := uiChecks + 1;
IF (fbTimer.udiElapsedMs <> 100) OR NOT fbTimer.xDone THEN
    uiFailures := uiFailures + 1;
END_IF;
fbTimer(xReset := TRUE, xEnable := TRUE, xQualified := TRUE,
    udiDeltaMs := 100, udiTargetMs := 100);
uiChecks := uiChecks + 1;
IF (fbTimer.udiElapsedMs <> 0) OR fbTimer.xDone THEN
    uiFailures := uiFailures + 1;
END_IF;
fbTimer(xReset := FALSE, xEnable := TRUE, xQualified := TRUE,
    udiDeltaMs := 100, udiTargetMs := 0);
uiChecks := uiChecks + 1;
IF (fbTimer.udiElapsedMs <> 0) OR fbTimer.xDone THEN
    uiFailures := uiFailures + 1;
END_IF;

// 03 - Structural recipe validation. Physical limits need adapter tests.
stRecipe.udiRecipeID := 1;
stRecipe.udiRevision := 1;
stRecipe.uiStepCount := 2;
FOR uiIndex := 1 TO 2 DO
    stRecipe.astSteps[uiIndex].uiStepID := uiIndex;
    stRecipe.astSteps[uiIndex].uiPhaseID := 1;
    stRecipe.astSteps[uiIndex].uiProfileID := 1;
    stRecipe.astSteps[uiIndex].eKind := E_SEQ_STEP_KIND.WaitQualified;
    stRecipe.astSteps[uiIndex].udiQualifiedMs := 100;
    stRecipe.astSteps[uiIndex].udiTimeoutMs := 200;
END_FOR;
fbRecipe(stRecipe := stRecipe);
uiChecks := uiChecks + 1;
IF NOT fbRecipe.xValid OR (fbRecipe.uiInvalidStep <> 0)
   OR (fbRecipe.eReason <> E_SEQ_REASON.None) THEN
    uiFailures := uiFailures + 1;
END_IF;
stRecipe.astSteps[2].uiStepID := 1;
fbRecipe(stRecipe := stRecipe);
uiChecks := uiChecks + 1;
IF fbRecipe.xValid OR (fbRecipe.uiInvalidStep <> 2)
   OR (fbRecipe.eReason <> E_SEQ_REASON.RecipeInvalid) THEN
    uiFailures := uiFailures + 1;
END_IF;
stRecipe.astSteps[2].uiStepID := 2;
stRecipe.uiStepCount := 0;
fbRecipe(stRecipe := stRecipe);
uiChecks := uiChecks + 1;
IF fbRecipe.xValid OR (fbRecipe.uiInvalidStep <> 0) THEN
    uiFailures := uiFailures + 1;
END_IF;
stRecipe.uiStepCount := 17;
fbRecipe(stRecipe := stRecipe);
uiChecks := uiChecks + 1;
IF fbRecipe.xValid OR (fbRecipe.uiInvalidStep <> 0) THEN
    uiFailures := uiFailures + 1;
END_IF;
stRecipe.uiStepCount := UINT#65535;
fbRecipe(stRecipe := stRecipe);
uiChecks := uiChecks + 1;
IF fbRecipe.xValid OR (fbRecipe.uiInvalidStep <> 0) THEN
    uiFailures := uiFailures + 1;
END_IF;
stRecipe.uiStepCount := 2;
stRecipe.udiRevision := 0;
fbRecipe(stRecipe := stRecipe);
uiChecks := uiChecks + 1;
IF fbRecipe.xValid OR (fbRecipe.uiInvalidStep <> 0) THEN
    uiFailures := uiFailures + 1;
END_IF;
stRecipe.udiRevision := 1;
stRecipe.astSteps[2].uiProfileID := 0;
fbRecipe(stRecipe := stRecipe);
uiChecks := uiChecks + 1;
IF fbRecipe.xValid OR (fbRecipe.uiInvalidStep <> 2) THEN
    uiFailures := uiFailures + 1;
END_IF;
stRecipe.astSteps[2].uiProfileID := 1;
stRecipe.astSteps[2].udiQualifiedMs := 201;
fbRecipe(stRecipe := stRecipe);
uiChecks := uiChecks + 1;
IF fbRecipe.xValid OR (fbRecipe.uiInvalidStep <> 2) THEN
    uiFailures := uiFailures + 1;
END_IF;
stRecipe.astSteps[2].udiQualifiedMs := 0;
fbRecipe(stRecipe := stRecipe);
uiChecks := uiChecks + 1;
IF fbRecipe.xValid OR (fbRecipe.uiInvalidStep <> 2) THEN
    uiFailures := uiFailures + 1;
END_IF;
stRecipe.astSteps[2].udiQualifiedMs := 200;
fbRecipe(stRecipe := stRecipe);
uiChecks := uiChecks + 1;
IF NOT fbRecipe.xValid THEN uiFailures := uiFailures + 1; END_IF;

// 04 - Ring wrap, full queue drop-new, exact ACK and repeated ACK.
stEvent.udiSessionID := 1;
stEvent.uiProcessID := 1;
stEvent.udiEventID := 900; // Producer ID must be overwritten by the queue.
FOR uiIndex := 1 TO 32 DO
    fbQueue(xPush := TRUE, stEvent := stEvent, udiAckEventID := 0);
END_FOR;
uiChecks := uiChecks + 1;
IF (fbQueue.uiCount <> 32) OR (fbQueue.stHead.udiEventID <> 1)
   OR NOT fbQueue.xAvailable OR (fbQueue.udiDropped <> 0) THEN
    uiFailures := uiFailures + 1;
END_IF;
fbQueue(xPush := TRUE, stEvent := stEvent, udiAckEventID := 0);
uiChecks := uiChecks + 1;
IF (fbQueue.uiCount <> 32) OR (fbQueue.stHead.udiEventID <> 1)
   OR (fbQueue.udiDropped <> 1) THEN
    uiFailures := uiFailures + 1;
END_IF;
fbQueue(xPush := FALSE, stEvent := stEvent, udiAckEventID := 1);
uiChecks := uiChecks + 1;
IF (fbQueue.uiCount <> 31) OR (fbQueue.stHead.udiEventID <> 2) THEN
    uiFailures := uiFailures + 1;
END_IF;
fbQueue(xPush := FALSE, stEvent := stEvent, udiAckEventID := 1);
fbQueue(xPush := FALSE, stEvent := stEvent, udiAckEventID := 100);
uiChecks := uiChecks + 1;
IF (fbQueue.uiCount <> 31) OR (fbQueue.stHead.udiEventID <> 2) THEN
    uiFailures := uiFailures + 1;
END_IF;
// Pop then push; accepted new event gets ID33 (dropped event consumed no ID).
fbQueue(xPush := TRUE, stEvent := stEvent, udiAckEventID := 2);
fbQueue(xPush := TRUE, stEvent := stEvent, udiAckEventID := 0);
uiChecks := uiChecks + 1;
IF (fbQueue.uiCount <> 32) OR (fbQueue.stHead.udiEventID <> 3) THEN
    uiFailures := uiFailures + 1;
END_IF;
xDrainCorrect := TRUE;
FOR udiExpectedID := 3 TO 34 DO
    IF NOT fbQueue.xAvailable OR (fbQueue.stHead.udiEventID <> udiExpectedID) THEN
        xDrainCorrect := FALSE;
    END_IF;
    fbQueue(xPush := FALSE, stEvent := stEvent, udiAckEventID := udiExpectedID);
END_FOR;
uiChecks := uiChecks + 1;
IF NOT xDrainCorrect OR fbQueue.xAvailable OR (fbQueue.uiCount <> 0)
   OR (fbQueue.stHead.udiEventID <> 0) THEN
    uiFailures := uiFailures + 1;
END_IF;
// A speculative ACK cannot remove the event first enqueued by this same call.
fbQueue(xPush := TRUE, stEvent := stEvent, udiAckEventID := 35);
uiChecks := uiChecks + 1;
IF NOT fbQueue.xAvailable OR (fbQueue.uiCount <> 1)
   OR (fbQueue.stHead.udiEventID <> 35) OR (fbQueue.udiDropped <> 1) THEN
    uiFailures := uiFailures + 1;
END_IF;

// 05 - Command high-water mark survives repeats, clear, old IDs, wrong sessions.
stCommand.xValid := TRUE;
stCommand.udiSessionID := 1;
stCommand.uiProcessID := 1;
stCommand.udiRequestID := 10;
stCommand.eCommand := E_SEQ_CMD.Start;
fbGate(stRequest := stCommand, udiSessionID := 1, uiProcessID := 1);
uiChecks := uiChecks + 1;
IF NOT fbGate.xNew OR (fbGate.eReason <> E_SEQ_REASON.None)
   OR (fbGate.udiLastRequestID <> 10) THEN
    uiFailures := uiFailures + 1;
END_IF;
fbGate(stRequest := stCommand, udiSessionID := 1, uiProcessID := 1);
uiChecks := uiChecks + 1;
IF fbGate.xNew THEN uiFailures := uiFailures + 1; END_IF;
stCommand.xValid := FALSE;
fbGate(stRequest := stCommand, udiSessionID := 1, uiProcessID := 1);
stCommand.xValid := TRUE;
fbGate(stRequest := stCommand, udiSessionID := 1, uiProcessID := 1);
uiChecks := uiChecks + 1;
IF fbGate.xNew OR (fbGate.udiLastRequestID <> 10) THEN
    uiFailures := uiFailures + 1;
END_IF;
stCommand.eCommand := E_SEQ_CMD.Stop;
fbGate(stRequest := stCommand, udiSessionID := 1, uiProcessID := 1);
uiChecks := uiChecks + 1;
IF fbGate.xNew THEN uiFailures := uiFailures + 1; END_IF;
stCommand.udiRequestID := 9;
fbGate(stRequest := stCommand, udiSessionID := 1, uiProcessID := 1);
uiChecks := uiChecks + 1;
IF NOT fbGate.xNew OR (fbGate.eReason <> E_SEQ_REASON.InvalidRequest)
   OR (fbGate.udiLastRequestID <> 10) THEN
    uiFailures := uiFailures + 1;
END_IF;
fbGate(stRequest := stCommand, udiSessionID := 1, uiProcessID := 1);
uiChecks := uiChecks + 1;
IF fbGate.xNew THEN uiFailures := uiFailures + 1; END_IF;
stCommand.udiRequestID := 10;
fbGate(stRequest := stCommand, udiSessionID := 1, uiProcessID := 1);
uiChecks := uiChecks + 1;
IF NOT fbGate.xNew OR (fbGate.eReason <> E_SEQ_REASON.InvalidRequest)
   OR (fbGate.udiLastRequestID <> 10) THEN
    uiFailures := uiFailures + 1;
END_IF;
stCommand.udiSessionID := 2;
stCommand.udiRequestID := 1000;
fbGate(stRequest := stCommand, udiSessionID := 1, uiProcessID := 1);
uiChecks := uiChecks + 1;
IF NOT fbGate.xNew OR (fbGate.eReason <> E_SEQ_REASON.SessionMismatch)
   OR (fbGate.udiLastRequestID <> 10) THEN
    uiFailures := uiFailures + 1;
END_IF;
stCommand.udiSessionID := 1;
stCommand.udiRequestID := 11;
fbGate(stRequest := stCommand, udiSessionID := 1, uiProcessID := 1);
uiChecks := uiChecks + 1;
IF NOT fbGate.xNew OR (fbGate.eReason <> E_SEQ_REASON.None)
   OR (fbGate.udiLastRequestID <> 11) THEN
    uiFailures := uiFailures + 1;
END_IF;
stCommand.uiProcessID := 2;
stCommand.udiRequestID := 12;
fbGate(stRequest := stCommand, udiSessionID := 1, uiProcessID := 1);
uiChecks := uiChecks + 1;
IF NOT fbGate.xNew OR (fbGate.eReason <> E_SEQ_REASON.WrongProcess)
   OR (fbGate.udiLastRequestID <> 12) THEN
    uiFailures := uiFailures + 1;
END_IF;
stCommand.uiProcessID := 1;
fbGate(stRequest := stCommand, udiSessionID := 1, uiProcessID := 1);
uiChecks := uiChecks + 1;
IF fbGate.xNew THEN uiFailures := uiFailures + 1; END_IF;
stCommand.udiRequestID := 13;
fbGate(stRequest := stCommand, udiSessionID := 1, uiProcessID := 1);
uiChecks := uiChecks + 1;
IF NOT fbGate.xNew OR (fbGate.eReason <> E_SEQ_REASON.None)
   OR (fbGate.udiLastRequestID <> 13) THEN
    uiFailures := uiFailures + 1;
END_IF;

xDone := TRUE;
END_PROGRAM

(* ---- PRG_SEQ_TraceEngineTests.st ---- *)
// Offline-only fixtures: no Control outputs, no physical I/O, no process Start.
// Call once per scan in an isolated simulation task. Reinitialize to run again.
// The clock values below are assertions used to exercise flags, not measured time.
PROGRAM PRG_SEQ_TraceEngineTests
VAR
    xDone : BOOL;
    uiTests : UINT;
    uiFailures : UINT;
    uiFirstFailure : UINT := UINT#65535;
    uiCase : UINT;
    xPass : BOOL;
    fbSeq : FB_Sequence;
    stCfg : ST_SEQ_CONFIG := (uiProcessID := 1, udiSessionID := 9,
        udiMaxFeedbackAgeMs := 250, udiTransitionTimeoutMs := 5000,
        udiMaxCycleMs := 100, uiMachineID := 2, uiProducerSourceID := 3);
    stClock : ST_SEQ_TRACE_TIME;
    stAuth : ST_SEQ_CONTROL_AUTHORITY;
    stCmd : ST_SEQ_COMMAND_REQUEST;
    stRecipe : ST_SEQ_RECIPE;
    udiAckSession : UDINT;
    udiAckID : UDINT;
END_VAR

IF xDone THEN RETURN; END_IF;
stAuth.xValid := TRUE;
stAuth.udiSessionID := 9;
stAuth.uiProcessID := 1;
stAuth.udiAuthorityID := 1;
stAuth.xAllowRequests := TRUE;
stAuth.xAllowExecution := FALSE;
stAuth.xAllowPublication := TRUE;
stAuth.udiAgeMs := 0;
stClock.udiTickMs := 100 + UINT_TO_UDINT(uiCase) * 10;
stClock.xValid := uiCase <> 0;
stClock.xSynthetic := FALSE;
stCmd.xValid := FALSE;
udiAckSession := 9;
udiAckID := 0;

IF uiCase = 0 THEN
    stRecipe.udiRecipeID := 1;
    stRecipe.udiRevision := 1;
    stRecipe.uiStepCount := 1;
    stRecipe.astSteps[1].uiStepID := 10;
    stRecipe.astSteps[1].uiPhaseID := 20;
    stRecipe.astSteps[1].uiProfileID := 30;
    stRecipe.astSteps[1].eKind := E_SEQ_STEP_KIND.WaitComplete;
    stRecipe.astSteps[1].udiTimeoutMs := 1000;
    stCmd.udiSessionID := 9;
    stCmd.uiProcessID := 1;
    stCmd.uiSourceID := 4;
    stCmd.udiRequestID := 1;
    stCmd.eCommand := E_SEQ_CMD.LoadRecipe;
    stCmd.udiRecipeID := 1;
    stCmd.udiRecipeRevision := 1;
END_IF;
CASE uiCase OF
1, 10: stCmd.xValid := TRUE;
2: stClock.xSynthetic := TRUE;
3: stClock.xValid := FALSE;
4: udiAckSession := 8; udiAckID := 1;
5, 6: udiAckID := 1;
7: stAuth.xAllowPublication := FALSE; udiAckID := 2;
9: udiAckID := 2;
29: udiAckID := 3;
31: stCfg.uiMachineID := 99;
32: stCfg.uiMachineID := 2;
END_CASE;
IF (uiCase >= 11) AND (uiCase <= 27) THEN
    stCmd.xValid := TRUE;
    stCmd.udiRequestID := UINT_TO_UDINT(uiCase);
    stCmd.udiRecipeID := 99; // Rejected reference; applied recipe stays 1.
END_IF;

fbSeq(xEnable := FALSE, stConfig := stCfg, udiDeltaMs := 10,
    stTraceTime := stClock, stCommand := stCmd, stRecipeCandidate := stRecipe,
    stAuthority := stAuth, udiEventAckSessionID := udiAckSession,
    udiEventAckID := udiAckID);
xPass := TRUE;
CASE uiCase OF
0:
    xPass := NOT fbSeq.stRuntime.xTimeValid AND NOT fbSeq.stRuntime.xTraceReady
        AND fbSeq.stRuntime.xTraceHistoryComplete AND (fbSeq.stRuntime.udiRevision = 1);
1:
    xPass := fbSeq.stRuntime.xTraceReady AND (fbSeq.uiEventCount = 2)
        AND (fbSeq.stEvent.eKind = E_SEQ_EVENT_KIND.RecipeLoaded)
        AND (fbSeq.stEvent.udiOccurrenceTickMs = 110)
        AND (fbSeq.stEvent.uiMachineID = 2) AND (fbSeq.stEvent.uiProducerSourceID = 3)
        AND (fbSeq.stEvent.uiSourceID = 4) AND (fbSeq.stEvent.udiRequestedRecipeID = 1);
2:
    xPass := fbSeq.stRuntime.xSyntheticTime AND NOT fbSeq.stRuntime.xTraceReady
        AND NOT fbSeq.stEvent.xSyntheticTime AND (fbSeq.stEvent.udiOccurrenceTickMs = 110);
3:
    xPass := NOT fbSeq.stRuntime.xTraceReady AND NOT fbSeq.stRuntime.xTimeValid
        AND fbSeq.stEvent.xOccurrenceTimeValid;
4:
    xPass := (fbSeq.stEvent.udiEventID = 1) AND (fbSeq.uiEventCount = 2);
5, 6:
    xPass := (fbSeq.stEvent.udiEventID = 2) AND (fbSeq.uiEventCount = 1);
7:
    xPass := NOT fbSeq.stRuntime.xDataValid AND NOT fbSeq.xEventAvailable
        AND (fbSeq.stEvent.udiEventID = 0) AND (fbSeq.uiEventCount = 0);
8:
    xPass := (fbSeq.stEvent.udiEventID = 2) AND (fbSeq.uiEventCount = 1);
9, 10:
    xPass := NOT fbSeq.xEventAvailable AND (fbSeq.uiEventCount = 0);
28:
    xPass := (fbSeq.uiEventCount = 32) AND (fbSeq.udiEventsDropped = 2)
        AND NOT fbSeq.stRuntime.xTraceHistoryComplete AND NOT fbSeq.stRuntime.xTraceReady
        AND (fbSeq.stEvent.udiEventID = 3) AND (fbSeq.stEvent.udiOccurrenceTickMs = 210)
        AND (fbSeq.stEvent.udiRecipeID = 1) AND (fbSeq.stEvent.udiRequestedRecipeID = 99);
29, 30:
    xPass := (fbSeq.uiEventCount = 31) AND (fbSeq.udiEventsDropped = 2)
        AND NOT fbSeq.stRuntime.xTraceHistoryComplete AND NOT fbSeq.stRuntime.xTraceReady
        AND (fbSeq.stEvent.udiEventID = 4);
31:
    xPass := NOT fbSeq.stRuntime.xDataValid AND NOT fbSeq.xEventAvailable
        AND NOT fbSeq.stControlRequest.xValid;
32:
    xPass := (fbSeq.stRuntime.eState = E_SEQ_STATE.Faulted)
        AND (fbSeq.stRuntime.eReason = E_SEQ_REASON.ConfigInvalid)
        AND NOT fbSeq.stRuntime.xTraceHistoryComplete
        AND (fbSeq.uiEventCount = 32) AND (fbSeq.udiEventsDropped = 3)
        AND (fbSeq.stEvent.udiEventID = 4);
END_CASE;
IF (uiCase >= 11) AND (uiCase <= 27) THEN
    xPass := (fbSeq.stCommandResult.eResult = E_SEQ_RESULT.Rejected)
        AND (fbSeq.stRuntime.udiRecipeID = 1) AND (fbSeq.stRuntime.eState = E_SEQ_STATE.Idle);
END_IF;
uiTests := uiTests + 1;
IF NOT xPass THEN
    uiFailures := uiFailures + 1;
    IF uiFirstFailure = UINT#65535 THEN uiFirstFailure := uiCase; END_IF;
END_IF;
IF uiCase = 32 THEN xDone := TRUE; ELSE uiCase := uiCase + 1; END_IF;
END_PROGRAM

(* ---- PRG_SEQ_TraceTests.st ---- *)
// OFFLINE EVENT-BUILDER FIXTURES ONLY. No Service, transport or physical I/O.
// Run cyclically in the simulator. Expected xDone/uiChecks/uiFailures/
// uiFirstFailureStep = TRUE/16/0/65535 after 16 scans. Native run is required;
// a static source check does not establish that these assertions have passed.
PROGRAM PRG_SEQ_TraceTests
VAR
    fbBuilder : FB_SEQ_EventBuilder;
    stBefore : ST_SEQ_RUNTIME;
    stAfter : ST_SEQ_RUNTIME;
    stCommand : ST_SEQ_COMMAND_REQUEST;
    stResult : ST_SEQ_COMMAND_RESULT;
    stEmptyRuntime : ST_SEQ_RUNTIME;
    stEmptyCommand : ST_SEQ_COMMAND_REQUEST;
    stEmptyResult : ST_SEQ_COMMAND_RESULT;
    xCommandNew : BOOL;
    xRecipeLoaded : BOOL;
    xStepCompleted : BOOL;
    xConfirmed : BOOL;
    xPass : BOOL;
    i : UINT;
    uiStep : UINT;
    uiChecks : UINT;
    uiFailures : UINT;
    uiFirstFailureStep : UINT := UINT#65535;
    xDone : BOOL;
END_VAR

IF xDone THEN RETURN; END_IF;
// Each fixture is independent, but the same builder instance is reused to
// detect stale outputs. DataValid remains FALSE: inputs are internal snapshots.
stBefore := stEmptyRuntime;
stBefore.uiMachineID := 2;
stBefore.uiProducerSourceID := 31;
stBefore.uiProcessID := 4;
stBefore.udiSessionID := 9001;
stBefore.udiAuthorityID := 6;
stBefore.udiRecipeID := 17;
stBefore.udiRecipeRevision := 3;
stBefore.udiBatchID := 81;
stBefore.eState := E_SEQ_STATE.Running;
stBefore.uiStepID := 100;
stBefore.uiPhaseID := 10;
stBefore.uiProfileID := 20;
stBefore.udiLastControlIntentID := 301;
stBefore.udiTickMs := 240;
stBefore.xTimeValid := TRUE;
stBefore.xSyntheticTime := TRUE;
stAfter := stBefore;
stAfter.udiTickMs := 250;
stAfter.udiLastControlIntentID := 302;
stCommand := stEmptyCommand;
stCommand.udiSessionID := 9001;
stCommand.udiRequestID := 25;
stCommand.uiSourceID := 7;
stCommand.uiProcessID := 4;
stResult := stEmptyResult;
stResult.udiSessionID := 9001;
stResult.udiRequestID := 25;
stResult.uiSourceID := 7;
stResult.uiProcessID := 4;
xCommandNew := FALSE;
xRecipeLoaded := FALSE;
xStepCompleted := FALSE;
xConfirmed := FALSE;

CASE uiStep OF
0, 14:
    // Quiet Idle before/after, including after a nonempty event-producing scan.
    stBefore.eState := E_SEQ_STATE.Idle;
    stAfter := stBefore;
1:
    // Reset clears runtime identity but must retain the prior lot in the facts.
    stBefore.eState := E_SEQ_STATE.Faulted;
    stBefore.eReason := E_SEQ_REASON.StepTimeout;
    stAfter.eState := E_SEQ_STATE.Idle;
    stAfter.uiStepID := 0;
    stAfter.udiBatchID := 0;
2:
    // Reject candidate 999; do not report it as the already applied recipe 17.
    xCommandNew := TRUE;
    stCommand.eCommand := E_SEQ_CMD.LoadRecipe;
    stCommand.udiRecipeID := 999;
    stCommand.udiRecipeRevision := 5;
    stResult.xValid := TRUE;
    stResult.eCommand := E_SEQ_CMD.LoadRecipe;
    stResult.eResult := E_SEQ_RESULT.Rejected;
    stResult.eReason := E_SEQ_REASON.InvalidRecipeRef;
    stAfter.xTimeValid := FALSE;
3:
    // Timing arguments include the completion scan before the core resets them.
    stBefore.udiPromptID := 54;
    stAfter.uiStepID := 200;
    stAfter.uiPhaseID := 11;
    stAfter.uiProfileID := 21;
    stAfter.udiStepElapsedMs := 0;
    stAfter.udiQualifiedElapsedMs := 0;
    xStepCompleted := TRUE;
4:
    // A fault is not a successful/aborted/stopped batch terminal outcome.
    stAfter.eState := E_SEQ_STATE.Faulted;
    stAfter.eReason := E_SEQ_REASON.ResourceLost;
5:
    stBefore.eState := E_SEQ_STATE.Starting;
    stAfter.udiResourceToken := 77;
6:
    // Resume keeps PromptID: no repeated PromptIssued or StepStarted.
    stBefore.eState := E_SEQ_STATE.Held;
    stBefore.udiPromptID := 55;
    stBefore.xWaitingOperator := FALSE;
    stAfter.udiPromptID := 55;
    stAfter.xWaitingOperator := TRUE;
7:
    stBefore.udiPromptID := 54;
    stAfter.udiPromptID := 55;
    stAfter.xWaitingOperator := TRUE;
8:
    stBefore.udiPromptID := 55;
    stBefore.xWaitingOperator := TRUE;
    stAfter.udiPromptID := 0;
    stAfter.uiStepID := 200;
    stAfter.uiPhaseID := 11;
    stAfter.uiProfileID := 21;
    xCommandNew := TRUE;
    xConfirmed := TRUE;
    xStepCompleted := TRUE;
    stCommand.eCommand := E_SEQ_CMD.ConfirmStep;
    stCommand.udiPromptID := 55;
    stCommand.uiStepID := 100;
    stResult.xValid := TRUE;
    stResult.eCommand := E_SEQ_CMD.ConfirmStep;
    stResult.eResult := E_SEQ_RESULT.Accepted;
9:
    stBefore.eState := E_SEQ_STATE.Completing;
    stBefore.udiResourceToken := 77;
    stAfter.eState := E_SEQ_STATE.Complete;
10:
    stBefore.eState := E_SEQ_STATE.Stopping;
    stAfter.eState := E_SEQ_STATE.Stopped;
11:
    stBefore.eState := E_SEQ_STATE.Aborting;
    stAfter.eState := E_SEQ_STATE.Aborted;
12:
    stBefore.eState := E_SEQ_STATE.Idle;
    stBefore.udiRecipeID := 0;
    stBefore.udiRecipeRevision := 0;
    stAfter.eState := E_SEQ_STATE.Idle;
    stAfter.xRecipeLoaded := TRUE;
    xRecipeLoaded := TRUE;
    xCommandNew := TRUE;
    stCommand.eCommand := E_SEQ_CMD.LoadRecipe;
    stCommand.udiRecipeID := 17;
    stCommand.udiRecipeRevision := 3;
    stResult.xValid := TRUE;
    stResult.eCommand := E_SEQ_CMD.LoadRecipe;
    stResult.eResult := E_SEQ_RESULT.Accepted;
13:
    stBefore.eState := E_SEQ_STATE.Idle;
    stBefore.udiBatchID := 0;
    stBefore.uiStepID := 0;
    stAfter.eState := E_SEQ_STATE.Starting;
    xCommandNew := TRUE;
    stCommand.eCommand := E_SEQ_CMD.Start;
    stCommand.udiBatchID := 81;
    stResult.xValid := TRUE;
    stResult.eCommand := E_SEQ_CMD.Start;
    stResult.eResult := E_SEQ_RESULT.Accepted;
15:
    // Replacement token records both identities, not just the new token.
    stBefore.udiResourceToken := 77;
    stAfter.udiResourceToken := 78;
    stAfter.udiAuthorityID := 7;
END_CASE;

fbBuilder(stBefore := stBefore, stAfter := stAfter,
    stCommand := stCommand, stResult := stResult,
    xCommandNew := xCommandNew, xRecipeLoaded := xRecipeLoaded,
    xStepCompleted := xStepCompleted, xConfirmed := xConfirmed,
    udiCompletedStepElapsedMs := 1010, udiCompletedQualifiedMs := 800);

xPass := FALSE;
CASE uiStep OF
0, 14:
    xPass := fbBuilder.uiCount = 0;
    FOR i := 1 TO 16 DO
        xPass := xPass AND (fbBuilder.astEvents[i].udiSessionID = 0)
            AND (fbBuilder.astEvents[i].udiRequestID = 0)
            AND (fbBuilder.astEvents[i].udiBatchID = 0);
    END_FOR;
1:
    xPass := (fbBuilder.uiCount = 3)
        AND (fbBuilder.astEvents[1].eKind = E_SEQ_EVENT_KIND.StateChanged)
        AND (fbBuilder.astEvents[1].eStateBefore = E_SEQ_STATE.Faulted)
        AND (fbBuilder.astEvents[1].eState = E_SEQ_STATE.Idle)
        AND (fbBuilder.astEvents[1].udiBatchID = 81)
        AND (fbBuilder.astEvents[1].udiBatchIDBefore = 81)
        AND (fbBuilder.astEvents[1].uiStepIDBefore = 100)
        AND (fbBuilder.astEvents[1].udiRecipeIDBefore = 17)
        AND (fbBuilder.astEvents[3].eKind = E_SEQ_EVENT_KIND.FaultCleared)
        AND (fbBuilder.astEvents[3].eReason = E_SEQ_REASON.StepTimeout);
2:
    xPass := (fbBuilder.uiCount = 2)
        AND (fbBuilder.astEvents[1].eKind = E_SEQ_EVENT_KIND.CommandResult)
        AND (fbBuilder.astEvents[2].eKind = E_SEQ_EVENT_KIND.RecipeRejected)
        AND (fbBuilder.astEvents[2].udiRecipeID = 17)
        AND (fbBuilder.astEvents[2].udiRequestedRecipeID = 999)
        AND (fbBuilder.astEvents[2].udiRequestedRecipeRevision = 5)
        AND (fbBuilder.astEvents[2].udiRequestID = 25)
        AND (fbBuilder.astEvents[2].uiSourceID = 7)
        AND (fbBuilder.astEvents[2].uiProducerSourceID = 31)
        AND (fbBuilder.astEvents[2].udiOccurrenceTickMs = 250)
        AND NOT fbBuilder.astEvents[2].xOccurrenceTimeValid
        AND fbBuilder.astEvents[2].xSyntheticTime;
3:
    xPass := (fbBuilder.uiCount = 3)
        AND (fbBuilder.astEvents[1].eKind = E_SEQ_EVENT_KIND.StepChanged)
        AND (fbBuilder.astEvents[2].eKind = E_SEQ_EVENT_KIND.StepFinished)
        AND (fbBuilder.astEvents[2].uiStepID = 100)
        AND (fbBuilder.astEvents[2].uiPhaseID = 10)
        AND (fbBuilder.astEvents[2].uiProfileID = 20)
        AND (fbBuilder.astEvents[2].udiIntentID = 301)
        AND (fbBuilder.astEvents[2].udiPromptID = 54)
        AND (fbBuilder.astEvents[2].udiStepElapsedMs = 1010)
        AND (fbBuilder.astEvents[2].udiQualifiedElapsedMs = 800)
        AND (fbBuilder.astEvents[3].eKind = E_SEQ_EVENT_KIND.StepStarted)
        AND (fbBuilder.astEvents[3].uiStepID = 200)
        AND (fbBuilder.astEvents[3].udiIntentID = 302);
4:
    xPass := (fbBuilder.uiCount = 2)
        AND (fbBuilder.astEvents[1].eKind = E_SEQ_EVENT_KIND.StateChanged)
        AND (fbBuilder.astEvents[2].eKind = E_SEQ_EVENT_KIND.FaultRaised)
        AND (fbBuilder.astEvents[2].eReason = E_SEQ_REASON.ResourceLost);
5:
    xPass := (fbBuilder.uiCount = 3)
        AND (fbBuilder.astEvents[2].eKind = E_SEQ_EVENT_KIND.StepStarted)
        AND (fbBuilder.astEvents[3].eKind = E_SEQ_EVENT_KIND.ResourceAcquired)
        AND (fbBuilder.astEvents[3].udiIntentID = 301)
        AND (fbBuilder.astEvents[3].udiResourceToken = 77)
        AND (fbBuilder.astEvents[3].udiResourceTokenBefore = 0);
6:
    xPass := (fbBuilder.uiCount = 1)
        AND (fbBuilder.astEvents[1].eKind = E_SEQ_EVENT_KIND.StateChanged);
7:
    xPass := (fbBuilder.uiCount = 1)
        AND (fbBuilder.astEvents[1].eKind = E_SEQ_EVENT_KIND.PromptIssued)
        AND (fbBuilder.astEvents[1].udiPromptID = 55);
8:
    xPass := (fbBuilder.uiCount = 5)
        AND (fbBuilder.astEvents[5].eKind = E_SEQ_EVENT_KIND.PromptConfirmed)
        AND (fbBuilder.astEvents[5].udiPromptID = 55)
        AND (fbBuilder.astEvents[5].udiRequestedPromptID = 55)
        AND (fbBuilder.astEvents[5].uiRequestedStepID = 100)
        AND (fbBuilder.astEvents[5].uiStepID = 100)
        AND (fbBuilder.astEvents[5].uiPhaseID = 10)
        AND (fbBuilder.astEvents[5].uiProfileID = 20)
        AND (fbBuilder.astEvents[5].udiIntentID = 301)
        AND (fbBuilder.astEvents[5].udiStepElapsedMs = 1010)
        AND (fbBuilder.astEvents[5].udiQualifiedElapsedMs = 800);
9:
    xPass := (fbBuilder.uiCount = 3)
        AND (fbBuilder.astEvents[2].eKind = E_SEQ_EVENT_KIND.BatchFinished)
        AND (fbBuilder.astEvents[2].eState = E_SEQ_STATE.Complete)
        AND (fbBuilder.astEvents[3].eKind = E_SEQ_EVENT_KIND.ResourceReleased)
        AND (fbBuilder.astEvents[3].udiIntentID = 301)
        AND (fbBuilder.astEvents[3].udiResourceToken = 77);
10:
    xPass := (fbBuilder.uiCount = 2)
        AND (fbBuilder.astEvents[2].eKind = E_SEQ_EVENT_KIND.BatchFinished)
        AND (fbBuilder.astEvents[2].eState = E_SEQ_STATE.Stopped);
11:
    xPass := (fbBuilder.uiCount = 2)
        AND (fbBuilder.astEvents[2].eKind = E_SEQ_EVENT_KIND.BatchFinished)
        AND (fbBuilder.astEvents[2].eState = E_SEQ_STATE.Aborted);
12:
    xPass := (fbBuilder.uiCount = 2)
        AND (fbBuilder.astEvents[1].eKind = E_SEQ_EVENT_KIND.RecipeLoaded)
        AND (fbBuilder.astEvents[2].eKind = E_SEQ_EVENT_KIND.CommandResult)
        AND (fbBuilder.astEvents[1].udiRecipeID = 17)
        AND (fbBuilder.astEvents[1].udiRecipeIDBefore = 0)
        AND (fbBuilder.astEvents[1].udiRequestID = 25);
13:
    xPass := (fbBuilder.uiCount = 4)
        AND (fbBuilder.astEvents[1].eKind = E_SEQ_EVENT_KIND.StateChanged)
        AND (fbBuilder.astEvents[2].eKind = E_SEQ_EVENT_KIND.StepChanged)
        AND (fbBuilder.astEvents[3].eKind = E_SEQ_EVENT_KIND.CommandResult)
        AND (fbBuilder.astEvents[4].eKind = E_SEQ_EVENT_KIND.BatchStarted)
        AND (fbBuilder.astEvents[4].eState = E_SEQ_STATE.Starting)
        AND (fbBuilder.astEvents[4].udiRequestedBatchID = 81);
15:
    xPass := (fbBuilder.uiCount = 2)
        AND (fbBuilder.astEvents[1].eKind = E_SEQ_EVENT_KIND.ResourceReleased)
        AND (fbBuilder.astEvents[1].udiResourceToken = 77)
        AND (fbBuilder.astEvents[1].udiAuthorityID = 6)
        AND (fbBuilder.astEvents[1].udiIntentID = 301)
        AND (fbBuilder.astEvents[2].eKind = E_SEQ_EVENT_KIND.ResourceAcquired)
        AND (fbBuilder.astEvents[2].udiResourceToken = 78)
        AND (fbBuilder.astEvents[2].udiAuthorityID = 7)
        AND (fbBuilder.astEvents[2].udiIntentID = 301);
END_CASE;
// Every emitted fact has source metadata, no fabricated wall-clock/EventID.
FOR i := 1 TO fbBuilder.uiCount DO
    xPass := xPass AND (fbBuilder.astEvents[i].udiEventID = 0)
        AND (fbBuilder.astEvents[i].uiContractMinor = 2)
        AND (fbBuilder.astEvents[i].uiMachineID = 2)
        AND (fbBuilder.astEvents[i].udiSessionID = 9001);
END_FOR;
uiChecks := uiChecks + 1;
IF NOT xPass THEN
    uiFailures := uiFailures + 1;
    IF uiFirstFailureStep = UINT#65535 THEN uiFirstFailureStep := uiStep; END_IF;
END_IF;
IF uiStep >= 15 THEN xDone := TRUE;
ELSE uiStep := uiStep + 1; END_IF;
END_PROGRAM
